FUNCTION TryConvert_TOD_TO_WORD : BOOL
VAR_INPUT
	in : TOD;
	out : REFERENCE TO WORD;
END_VAR

IF in > DatatypeLimits.MAX_VALUE_OF_TOD_WHICH_CAN_BE_HELD_IN_A_WORD THEN
	RETURN;
END_IF

out := TOD_TO_WORD(in);
TryConvert_TOD_TO_WORD := TRUE;

END_FUNCTION

(* stored: Version 1.1.0.1, ProductVersion 3.1.4024.12
   POU TryConvert_TOD_TO_WORD: Id {90c1b019-3b60-4866-975e-49da907f0fb9}, SpecialFunc None *)
